(* IEC 61131-3 sources: volt/packages/volt-lsp-iec/test-corpus/bakon-nano/Device/Plc Logic/Application/Library Manager/SysTarget, 18 files *)

(* ---- DEVICETYPES.gvl ---- *)
VAR_GLOBAL
	SYSTARGET_TYPE_SPECIAL_UNREGISTERED_SLOT : DWORD := 16#0;
	SYSTARGET_TYPE_PROGRAMMABLE : DWORD := 16#1000;
	SYSTARGET_TYPE_3S_SPECIAL_DEVICE : DWORD := 16#1001;
	SYSTARGET_TYPE_SAFETY_DEVICE : DWORD := 16#1002;
	SYSTARGET_TYPE_DRIVE : DWORD := 16#1003;
	SYSTARGET_TYPE_PARAMETRIZABLE : DWORD := 16#1004;
	SYSTARGET_TYPE_HMI : DWORD := 16#1005;
	SYSTARGET_TYPE_3S_SOFTMOTION : DWORD := 16#1006;
	SYSTARGET_TYPE_COMMUNICATION : DWORD := 16#1007;
END_VAR

(* ---- OPERATINGSYSTEMID.gvl ---- *)
VAR_GLOBAL
	SYSTARGET_OS_NONE : UDINT := 1;
	SYSTARGET_OS_WINDOWS : UDINT := 2;
	SYSTARGET_OS_WINDOWS_KERNEL : UDINT := 3;
	SYSTARGET_OS_WINDOWS_RTE : UDINT := 3;
	SYSTARGET_OS_WINDOWS_CE : UDINT := 4;
	SYSTARGET_OS_LINUX : UDINT := 5;
	SYSTARGET_OS_VXWORKS : UDINT := 6;
	SYSTARGET_OS_QNX : UDINT := 7;
	SYSTARGET_OS_UCOS : UDINT := 8;
END_VAR

(* ---- PROCESSORID.gvl ---- *)
VAR_GLOBAL
	TRG_X86 : UDINT := 1;
	TRG_ARM : UDINT := 2;
	TRG_PPC : UDINT := 3;
	TRG_MIPS : UDINT := 4;
	TRG_SH : UDINT := 5;
	TRG_BLACKFIN : UDINT := 6;
	TRG_TRICORE : UDINT := 7;
	TRG_NIOS : UDINT := 8;
	TRG_C16X : UDINT := 9;
	TRG_CORTEX : UDINT := 10;
	TRG_DSP : UDINT := 11;
	TRG_V850 : UDINT := 12;
	TRG_RX6 : UDINT := 13;
END_VAR

(* ---- SYSTARGETGETDEVICENAME.pou ---- *)
FUNCTION SYSTARGETGETDEVICENAME : RTS_IEC_RESULT
VAR_INPUT
	PWSZNAME : POINTER TO WSTRING;
	PNMAXLENGTH : POINTER TO UDINT;
END_VAR
END_FUNCTION

(* ---- SYSTARGETGETDEVICENAME2.pou ---- *)
FUNCTION SYSTARGETGETDEVICENAME2 : RTS_IEC_RESULT
VAR_INPUT
	PSZROUTERNAME : POINTER TO STRING;
	PWSZNAME : POINTER TO WSTRING;
	PNMAXLENGTH : POINTER TO UDINT;
END_VAR
END_FUNCTION

(* ---- SYSTARGETGETID.pou ---- *)
FUNCTION SYSTARGETGETID : RTS_IEC_RESULT
VAR_INPUT
	PULTARGETID : POINTER TO DWORD;
END_VAR
END_FUNCTION

(* ---- SYSTARGETGETID2.pou ---- *)
FUNCTION SYSTARGETGETID2 : RTS_IEC_RESULT
VAR_INPUT
	PSZROUTERNAME : POINTER TO STRING;
	PULTARGETID : POINTER TO DWORD;
END_VAR
END_FUNCTION

(* ---- SYSTARGETGETNODENAME.pou ---- *)
FUNCTION SYSTARGETGETNODENAME : RTS_IEC_RESULT
VAR_INPUT
	PWSZNAME : POINTER TO WSTRING;
	PNMAXLENGTH : POINTER TO UDINT;
END_VAR
END_FUNCTION

(* ---- SYSTARGETGETNODENAME2.pou ---- *)
FUNCTION SYSTARGETGETNODENAME2 : RTS_IEC_RESULT
VAR_INPUT
	PSZROUTERNAME : POINTER TO STRING;
	PWSZNAME : POINTER TO WSTRING;
	PNMAXLENGTH : POINTER TO UDINT;
END_VAR
END_FUNCTION

(* ---- SYSTARGETGETOPERATINGSYSTEMID.pou ---- *)
FUNCTION SYSTARGETGETOPERATINGSYSTEMID : RTS_IEC_RESULT
VAR_INPUT
	PUDIOPERATINGSYSTEMID : POINTER TO UDINT;
END_VAR
END_FUNCTION

(* ---- SYSTARGETGETPROCESSORID.pou ---- *)
FUNCTION SYSTARGETGETPROCESSORID : RTS_IEC_RESULT
VAR_INPUT
	PUDIPROCESSORID : POINTER TO UDINT;
END_VAR
END_FUNCTION

(* ---- SYSTARGETGETSERIALNUMBER.pou ---- *)
FUNCTION SYSTARGETGETSERIALNUMBER : RTS_IEC_RESULT
VAR_INPUT
	PPSSERIALNUMBER : POINTER TO POINTER TO STRING(255);
	PNMAXLEN : POINTER TO DINT;
END_VAR
END_FUNCTION

(* ---- SYSTARGETGETTYPE.pou ---- *)
FUNCTION SYSTARGETGETTYPE : RTS_IEC_RESULT
VAR_INPUT
	PULTYPE : POINTER TO DWORD;
END_VAR
END_FUNCTION

(* ---- SYSTARGETGETTYPE2.pou ---- *)
FUNCTION SYSTARGETGETTYPE2 : RTS_IEC_RESULT
VAR_INPUT
	PSZROUTERNAME : POINTER TO STRING;
	PULTYPE : POINTER TO DWORD;
END_VAR
END_FUNCTION

(* ---- SYSTARGETGETVENDORNAME.pou ---- *)
FUNCTION SYSTARGETGETVENDORNAME : RTS_IEC_RESULT
VAR_INPUT
	PWSZNAME : POINTER TO WSTRING;
	PNMAXLENGTH : POINTER TO UDINT;
END_VAR
END_FUNCTION

(* ---- SYSTARGETGETVENDORNAME2.pou ---- *)
FUNCTION SYSTARGETGETVENDORNAME2 : RTS_IEC_RESULT
VAR_INPUT
	PSZROUTERNAME : POINTER TO STRING;
	PWSZNAME : POINTER TO WSTRING;
	PNMAXLENGTH : POINTER TO UDINT;
END_VAR
END_FUNCTION

(* ---- SYSTARGETGETVERSION.pou ---- *)
FUNCTION SYSTARGETGETVERSION : RTS_IEC_RESULT
VAR_INPUT
	PULVERSION : POINTER TO DWORD;
END_VAR
END_FUNCTION

(* ---- SYSTARGETGETVERSION2.pou ---- *)
FUNCTION SYSTARGETGETVERSION2 : RTS_IEC_RESULT
VAR_INPUT
	PSZROUTERNAME : POINTER TO STRING;
	PULVERSION : POINTER TO DWORD;
END_VAR
END_FUNCTION
